	//Неисправности
	#T_notON_TON(
	             IN := (#sigOut AND NOT #OnSig AND NOT #Reset),
	             PT := #Set_T_notON
	);
	
	#notON := (#notON OR #T_notON_TON.Q) AND NOT #Reset;
	
	#T_notOFF_TON(
	             IN := (NOT #sigOut AND #OnSig AND NOT #Reset),
	             PT := #Set_T_notOFF
	);
	
	#notOFF := (#notOFF OR #T_notOFF_TON.Q) AND NOT #Reset;
	
	
	//Обобщенная неисправность
	#Fault := #notON OR #notOFF;
	
	//Авария
	#Alarm := (#Alarm OR #OnSig AND #sigOut AND NOT #Ready) AND NOT (#Reset);
	
	IF #DU THEN
	    #setSpeed := #setSpeedDU;
	ELSE
	    #setSpeed := #setSpeedAU;
	END_IF;
	
	#btnDU := false;
	
END_FUNCTION_BLOCK

FUNCTION_BLOCK "FB_IM1x1"
{ S7_Optimized_Access := 'FALSE' }
AUTHOR : Ivanez
VERSION : 0.1
//Абстактный механизм с 1й командой, 1й обратной связью (АУ, ДУ, МУ)
   VAR_INPUT 
      OnSig : Bool;   //      Сигнал сработавшего состояния
      OnCom : Bool;   //      Команда включения в автоматическом режиме
      Ready : Bool;   //      Условие готовности
      Reset : Bool;   //      Сброс
      btnAU : Bool;   //      Перевести в Автоматическое управление
      btnDU : Bool;   //      Перевести в Дистанционное управление
      prmDU : Bool;   //      Разрешение на перевод в ДУ
      btnDU_ON : Bool;   //      Включить в дистанционном управлении
      btnDU_OF : Bool;   //      Отключить в дистанционном управлении
      btnMU : Bool;   //      Перевести в местное управление
      btnMU_ON : Bool;   //      Включить в местном управлении
      btnMU_OF : Bool;   //      Отключить в местном управлении
      Set_T_notON : Time;   //      Задержа на формирование невключения
      Set_T_notOFF : Time;   //      Задержа на формирование неотключения
      setSpeedAU : Real;   //      Скорость в режиме автомат
      setSpeedDU : Real;   //      Скорость в режиме ДУoutputs
   END_VAR

   VAR_OUTPUT 
      AU : Bool;   //      Автоматическое управление (АУ)
      DU : Bool;   //      Дистанционное управление (ДУ)
      MU : Bool;   //      Местное управление (ДУ)
      notON : Bool;   //      Предупреждение о невключении
      notOFF : Bool;   //      Предупреждение о неотключении
      Alarm : Bool;   //      Авария (исчезновение готовности при работе)
      Fault : Bool;   //      Неисправность
      onOutFWD : Bool;   //      Сигнал на сработку механизма вперед
      PRM_btnDU_ON : Bool;   //      Разрешение кнопки включения в ДУ
      PRM_btnDU_OFF : Bool;   //      Разрешение кнопки отключения в ДУ
      setSpeed : Real;   //      скорость в автомате для частотникаvariables
   END_VAR

   VAR 
      sigOut : Bool;   //      Сигнал включения
      T_notON_TON {InstructionName := 'TON'; LibVersion := '1.0'; S7_SetPoint := 'False'} : TON;   //      Таймер невключения
      T_notOFF_TON {InstructionName := 'TON'; LibVersion := '1.0'; S7_SetPoint := 'False'} : TON;   //      Таймер неотключения
   END_VAR


BEGIN
	
	//Формирование автоматического управления
	IF #btnAU THEN
	    #AU := true;
	    #DU := false;
	    #MU := false;
	END_IF;
	//Формирование дистанционного управления 
	IF #btnDU THEN
	    #DU := true;
	    #AU := false;
	    #MU := false;
	END_IF;
	//Формирование местного управления
	IF #btnMU THEN
	    #MU := true;
	    #AU := false;
	    #DU := false;
	END_IF;
	
	IF NOT #AU AND NOT #DU AND NOT #MU THEN
	    #MU := true;
	END_IF;
	
	
	//Разрешения кнопок управления
	#PRM_btnDU_ON := (NOT #OnSig AND #DU OR #notON);
	#PRM_btnDU_OFF := ((#sigOut OR #OnSig) AND #DU OR #notOFF);
	
	
	//Формирование выходного сигнала
	#sigOut := #Ready AND ((#sigOut
	OR #AU AND #OnCom
	OR #DU AND #btnDU_ON
	OR #MU AND #btnMU_ON
	)
	AND NOT
	(#Alarm
	OR #AU AND NOT #OnCom
	OR #DU AND #btnDU_OF
	OR #MU AND #btnMU_OF
	OR #notON));
	
	#onOutFWD := #sigOut;
	
	//Неисправности
	#T_notON_TON(IN := (#sigOut AND NOT #OnSig AND NOT #Reset),
	             PT := #Set_T_notON
	);
	#notON := (#notON OR #T_notON_TON.Q) AND NOT #Reset;
	
	#T_notOFF_TON(IN := (NOT #sigOut AND #OnSig AND NOT #Reset),
	              PT := #Set_T_notOFF
	);
	#notOFF := (#notOFF OR #T_notOFF_TON.Q) AND NOT #Reset;
	
	//Обобщенная неисправность
	#Fault := #notON OR #notOFF;
	
	//Авария
	#Alarm := (#Alarm OR #OnSig AND #sigOut AND NOT #Ready) AND NOT (#Reset);
	
	IF #DU THEN
	    #setSpeed := #setSpeedDU;
	ELSE
	    #setSpeed := #setSpeedAU;
	END_IF;
	
END_FUNCTION_BLOCK

FUNCTION_BLOCK "FB_IM_Rout"
{ S7_Optimized_Access := 'FALSE' }
VERSION : 0.1
   VAR 
      M_321_Rollgang_Lift_PFM { S7_SetPoint := 'False'} : "FB_IM2x1";   // выкатной транспортер на лифте ПФМки
      M_322_Conveyor_2 : "FB_IM2x1";   // Выкатной транспортер после лифта
      M_324_Rout_Conveyor : "FB_IM2x1";   // выкатной транспортер последний
   END_VAR


BEGIN
	#M_321_Rollgang_Lift_PFM(OnSig:="DGI".F321K1_321K2,
	                         Ready:="ALG".Ready_Rout,
	                         Reset:="ALG".Reset OR "DGI".S76_2,
	                         btnAU:="ServDB".M_321.BtnAU OR "ALG".Auto_Sorting,
	                         btnDU:= "ServDB".M_321.BtnDU,
	                         prmDU:=TRUE,
	                         btnDU_ON:="ServDB".M_321.BtnFwd OR "ServDB".M_321.BtnBwd,
	                         btnDU_OF:="ServDB".M_321.BtnCmdStop,
	                         btnMU:="DGI".E88_3 OR "DGI".S88_2,
	                         btnMU_ON:="DGI".E88_3 OR "DGI".S88_2,
	                         btnMU_OF:=NOT ("DGI".E88_3 OR "DGI".S88_2),
	                         btn_Back_ON:= "ServDB".M_321.BtnBwd OR "DGI".S88_2,
	                         btn_Back_OFF:=NOT ("ServDB".M_321.BtnBwd OR "DGI".S88_2),
	                         Set_T_notON:=T#500ms,
	                         Set_T_notOFF:=T#500ms,
	                         AU=>"ServDB".M_321.AU,
	                         DU=>"ServDB".M_321.DU,
	                         MU=>"ServDB".M_321.MU,
	                         BACK=>"ServDB".M_321.BACK,
	                         Alarm=>"ServDB".M_321.Alarm,
	                         Fault=>"ServDB".M_321.Fault,
	                         onOutFWD=>"ServDB".M_321.CMD_ON,
	                         onOutBWD=>"ServDB".M_321.CMD_OFF,
	                         PRM_btnDU_ON=>"ServDB".M_321.PrmBtnDU_ON,
	                         PRM_btnDU_OFF=>"ServDB".M_321.PrmBtnDU_OF,
	                         PRMbtn_Back_ON=>"ServDB".M_321.PRMbtn_Back_ON,
	                         PRMbtn_Back_OFF=>"ServDB".M_321.PRMbtn_Back_OFF,
	                         setSpeed=>"ServDB".M_321.SetSpeed
	);
	
	"K1-321X1" := #M_321_Rollgang_Lift_PFM.onOutFWD AND "DGI".S16_1;
	"K1-321X1.1" := #M_321_Rollgang_Lift_PFM.onOutBWD AND "DGI".S16_1;
	
	
	
	#M_322_Conveyor_2(OnSig:="DGI".F322K1_322K2,
	                  Ready:="ALG".Ready_Rout,
	                  Reset:="ALG".Reset OR "DGI".S76_2,
	                  btnAU:="ServDB".M_322.BtnAU OR "ALG".Auto_Sorting,
	                  btnDU:="ServDB".M_322.BtnDU,
	                  prmDU:=TRUE,
	                  btnDU_ON:="ServDB".M_322.BtnFwd OR "ServDB".M_322.BtnBwd,
	                  btnDU_OF:="ServDB".M_322.BtnCmdStop,
	                  btnMU:= "DGI".S88_5 OR "DGI".S88_4,
	                  btnMU_ON:="DGI".S88_5 OR "DGI".S88_4,
	                  btnMU_OF:=NOT ("DGI".S88_5 OR "DGI".S88_4),
	                  btn_Back_ON:="ServDB".M_322.BtnBwd OR "DGI".S88_4,
	                  btn_Back_OFF:=NOT ("ServDB".M_322.BtnBwd OR "DGI".S88_4),
	                  Set_T_notON:=T#500ms,
	                  Set_T_notOFF:=T#500ms,
	                  AU=>"ServDB".M_322.AU,
	                  DU=>"ServDB".M_322.DU,
	                  MU=>"ServDB".M_322.MU,
	                  BACK=>"ServDB".M_322.BACK,
	                  Alarm=>"ServDB".M_322.Alarm,
	                  Fault=>"ServDB".M_322.Fault,
	                  onOutFWD=>"ServDB".M_322.CMD_ON,
	                  onOutBWD=>"ServDB".M_322.CMD_OFF,
	                  PRM_btnDU_ON=>"ServDB".M_322.PrmBtnDU_ON,
	                  PRM_btnDU_OFF=>"ServDB".M_322.PrmBtnDU_OF,
	                  PRMbtn_Back_ON=>"ServDB".M_322.PRMbtn_Back_ON,
	                  PRMbtn_Back_OFF=>"ServDB".M_322.PRMbtn_Back_OFF,
	                  setSpeed=>"ServDB".M_322.SetSpeed
	);
	
	
	"K1-322X1" := #M_322_Conveyor_2.onOutFWD;
	"K1-322X1.1" := #M_322_Conveyor_2.onOutBWD;
	
	#M_324_Rout_Conveyor(OnSig:="DGI".K1_324U1,
	                     Ready:="ALG".Ready_Rout,
	                     Reset:="ALG".Reset OR "DGI".S76_2,
	                     btnAU:= "ServDB".M_324.BtnAU OR "ALG".Auto_Sorting,
	                     btnDU:= "ServDB".M_324.BtnDU,
	                     prmDU:=TRUE,
	                     btnDU_ON:="ServDB".M_324.BtnFwd OR "ServDB".M_324.BtnBwd,
	                     btnDU_OF:="ServDB".M_324.BtnCmdStop,
	                     btnMU:= "DGI".S89_1 OR "DGI".S89_0,
	                     btnMU_ON:="DGI".S89_1 OR "DGI".S89_0,
	                     btnMU_OF:=NOT ("DGI".S89_1 OR "DGI".S89_0),
	                     btn_Back_ON:= "DGI".S89_0 OR "ServDB".M_324.BtnBwd,
	                     btn_Back_OFF:=NOT ("DGI".S89_0 OR "ServDB".M_324.BtnBwd),
	                     Set_T_notON:=T#1s,
	                     Set_T_notOFF:=T#2s,
	                     AU=>"ServDB".M_324.AU,
	                     DU=>"ServDB".M_324.DU,
	                     MU=>"ServDB".M_324.MU,
	                     BACK=>"ServDB".M_324.BACK,
	                     Alarm=>"ServDB".M_324.Alarm,
	                     Fault=>"ServDB".M_324.Fault,
	                     onOutFWD=>"ServDB".M_324.CMD_ON,
	                     onOutBWD=>"ServDB".M_324.CMD_OFF,
	                     PRM_btnDU_ON=>"ServDB".M_324.PrmBtnDU_ON,
	                     PRM_btnDU_OFF=>"ServDB".M_324.PrmBtnDU_OF,
	                     PRMbtn_Back_ON=>"ServDB".M_324.PRMbtn_Back_ON,
	                     PRMbtn_Back_OFF=>"ServDB".M_324.PRMbtn_Back_OFF,
	                     setSpeed=>"ServDB".M_324.SetSpeed
	);
	
	"K1-324U2" := #M_324_Rout_Conveyor.onOutFWD;
	"K1-324U2.2" := #M_324_Rout_Conveyor.onOutBWD;
	
END_FUNCTION_BLOCK

ORGANIZATION_BLOCK "PROG_ERR"   // OB121, LAD, ProgrammingError
TITLE = "Programming Error"
VERSION : 0.1
// stored: IsIECCheckEnabled false
   VAR_TEMP
      OB121_EV_CLASS : Byte;   // 16#25, Event class 2, Entering event state, Internal fault event
      OB121_SW_FLT : Byte;   // 16#XX Software programming fault
      OB121_PRIORITY : Byte;   // Priority of OB Execution
      OB121_OB_NUMBR : Byte;   // 121 (Organization block 121, OB121)
      OB121_BLK_TYPE : Byte;   // 16#88/8A/8B/8C/8E Type of block fault occured in
      OB121_RESERVED_1 : Byte;   // Reserved for system
      OB121_FLT_REG : Word;   // 16#XX Specific register that caused fault
      OB121_BLK_NUM : Word;   // Number of block that programming fault occured in
      OB121_PRG_ADDR : Word;   // Address in block where programming fault occured
      OB121_DATE_TIME : Date_And_Time;   // Date and time OB121 started
   END_VAR
BEGIN
END_ORGANIZATION_BLOCK

ORGANIZATION_BLOCK "BREAKUP ERROR"   // OB88, LAD, ProcessingInterrupt
TITLE = "Breakup Error"
VERSION : 0.1
// stored: IsIECCheckEnabled false
   VAR_TEMP
      OB88_EV_CLASS : Byte;   // 16#35 Event class 2, Entering event state, Internal fault event
      OB88_SW_FLT : Byte;   // 16#XX, Software programming fault
      OB88_PRIORITY : Byte;   // Priority of OB Execution
      OB88_OB_NUMBR : Byte;   // 88 (Organization block 88, OB88)
      OB88_BLK_TYPE : Byte;   // 16#88/8C/8E Type of block where breakup occured
      OB88_RESERVED_1 : Byte;   // Reserved for system
      OB88_FLT_PRIORITY : Byte;   // Priority of OB caused breakup
      OB88_FLT_OB_NUMBR : Byte;   // OB execution caused breakup
      OB88_BLK_NUM : Word;   // Number of block where breakup occured
      OB88_PRG_ADDR : Word;   // Address in block where breakup occured
      OB88_DATE_TIME : Date_And_Time;   // Date and time OB88 started
   END_VAR
BEGIN
END_ORGANIZATION_BLOCK

ORGANIZATION_BLOCK "COMM_FLT"   // OB87, LAD, CommunicationError
TITLE = "Communication Fault"
VERSION : 0.1
// stored: IsIECCheckEnabled false
   VAR_TEMP
      OB87_EV_CLASS : Byte;   // 16#39 Event class 3
      OB87_FLT_ID : Byte;   // 16#XX, Fault identifcation code
      OB87_PRIORITY : Byte;   // Priority of OB Execution
      OB87_OB_NUMBR : Byte;   // 87 (Organization block 87, OB87)
      OB87_RESERVED_1 : Byte;   // Reserved for system
      OB87_RESERVED_2 : Byte;   // Reserved for system
      OB87_RESERVED_3 : Word;   // Reserved for system
      OB87_RESERVED_4 : DWord;   // Reserved for system
      OB87_DATE_TIME : Date_And_Time;   // Date and time OB87 started
   END_VAR
BEGIN
END_ORGANIZATION_BLOCK

ORGANIZATION_BLOCK "CPU_FLT"   // OB84, LAD, CPUHardwareError
TITLE = "CPU Fault"
VERSION : 0.1
// stored: IsIECCheckEnabled false
   VAR_TEMP
      OB84_EV_CLASS : Byte;   // 16#38/39, Event class 3, module inserted/removed (8/9)
      OB84_FLT_ID : Byte;   // 16#81, Fault identifcation code
      OB84_PRIORITY : Byte;   // Priority of OB Execution
      OB84_OB_NUMBR : Byte;   // 84 (Organization block 84, OB84)
      OB84_RESERVED_1 : Byte;   // Reserved for system
      OB84_RESERVED_2 : Byte;   // Reserved for system
      OB84_RESERVED_3 : Word;   // Reserved for system
      OB84_RESERVED_4 : DWord;   // Reserved for system
      OB84_DATE_TIME : Date_And_Time;   // Date and time OB84 started
   END_VAR
BEGIN
END_ORGANIZATION_BLOCK

ORGANIZATION_BLOCK "CYCL_FLT"   // OB80, LAD, TimeErrorInterrupt
TITLE = "Cycle Time Fault"
VERSION : 0.1
// stored: IsIECCheckEnabled false
   VAR_TEMP
      OB80_EV_CLASS : Byte;   // 16#35, Event class 3, Entering event state, Internal fault event
      OB80_FLT_ID : Byte;   // 16#XX, Fault identifcation code
      OB80_PRIORITY : Byte;   // Priority of OB Execution
      OB80_OB_NUMBR : Byte;   // 80 (Organization block 80, OB80)
      OB80_RESERVED_1 : Byte;   // Reserved for system
      OB80_RESERVED_2 : Byte;   // Reserved for system
      OB80_ERROR_INFO : Word;   // Error information on event
      OB80_ERR_EV_CLASS : Byte;   // Class of event causing error
      OB80_ERR_EV_NUM : Byte;   // Number of event causing error
      OB80_OB_PRIORITY : Byte;   // Priority of OB causing error
      OB80_OB_NUM : Byte;   // Number of OB causing error
      OB80_DATE_TIME : Date_And_Time;   // Date and time OB80 started
   END_VAR
BEGIN
END_ORGANIZATION_BLOCK

ORGANIZATION_BLOCK "MOD_ERR"   // OB122, LAD, IOAccessError
TITLE = "Module Access Error"
VERSION : 0.1
// stored: IsIECCheckEnabled false
   VAR_TEMP
      OB122_EV_CLASS : Byte;   // 16#29, Event class 2, Entering event state, Internal fault event
      OB122_SW_FLT : Byte;   // 16#XX Software error code
      OB122_PRIORITY : Byte;   // Priority of OB Execution
      OB122_OB_NUMBR : Byte;   // 122 (Organization block 122, OB122)
      OB122_BLK_TYPE : Byte;   // 16#88/8C/8E Type of block fault occured in
      OB122_MEM_AREA : Byte;   // Memory area where access error occured
      OB122_MEM_ADDR : Word;   // Memory address where access error occured
      OB122_BLK_NUM : Word;   // Block number in which error occured
      OB122_PRG_ADDR : Word;   // Program address where error occured
      OB122_DATE_TIME : Date_And_Time;   // Date and time OB1 started
   END_VAR
BEGIN
END_ORGANIZATION_BLOCK

ORGANIZATION_BLOCK "OBNL_FLT"   // OB85, LAD, AccessError
TITLE = "Organization Block (OB) Not Loaded Fault"
VERSION : 0.1
// stored: IsIECCheckEnabled false
   VAR_TEMP
      OB85_EV_CLASS : Byte;   // 16#35 Event class 3
      OB85_FLT_ID : Byte;   // 16#XX, Fault identification code
      OB85_PRIORITY : Byte;   // Priority of OB Execution
      OB85_OB_NUMBR : Byte;   // 85 (Organization block 85, OB85)
      OB85_RESERVED_1 : Byte;   // Reserved for system
      OB85_RESERVED_2 : Byte;   // Reserved for system
      OB85_RESERVED_3 : Int;   // Reserved for system
      OB85_ERR_EV_CLASS : Byte;   // Class of event causing error
      OB85_ERR_EV_NUM : Byte;   // Number of event causing error
      OB85_OB_PRIOR : Byte;   // Priority of OB causing error
      OB85_OB_NUM : Byte;   // Number of OB causing error
      OB85_DATE_TIME : Date_And_Time;   // Date and time OB85 started
   END_VAR
BEGIN
END_ORGANIZATION_BLOCK

ORGANIZATION_BLOCK "PS_FLT"   // OB81, LAD, PowerSupplyError
TITLE = "Power Supply Fault"
VERSION : 0.1
// stored: IsIECCheckEnabled false
   VAR_TEMP
      OB81_EV_CLASS : Byte;   // 16#39, Event class 3, Entering event state, Internal fault event
      OB81_FLT_ID : Byte;   // 16#XX, Fault identifcation code
      OB81_PRIORITY : Byte;   // Priority of OB Execution
      OB81_OB_NUMBR : Byte;   // 81 (Organization block 81, OB81)
      OB81_RESERVED_1 : Byte;   // Reserved for system
      OB81_RESERVED_2 : Byte;   // Reserved for system
      OB81_RACK_CPU : Word;   // Bits 0 to 2: Rack no; Bit 3: 0=standby CPU, 1=master CPU; Bits 4 to 7: 1111
      OB81_RESERVED_3 : Byte;   // Reserved for system
      OB81_RESERVED_4 : Byte;   // Reserved for system
      OB81_RESERVED_5 : Byte;   // Reserved for system
      OB81_RESERVED_6 : Byte;   // Reserved for system
      OB81_DATE_TIME : Date_And_Time;   // Date and time OB81 started
   END_VAR
BEGIN
END_ORGANIZATION_BLOCK

ORGANIZATION_BLOCK "RACK_FLT"   // OB86, LAD, RackOrStationFailure
TITLE = "Loss Of Rack Fault"
VERSION : 0.1
// stored: IsIECCheckEnabled false
   VAR_TEMP
      OB86_EV_CLASS : Byte;   // 16#38/39 Event class 3
      OB86_FLT_ID : Byte;   // 16#C1/C4/C5, Fault identification code
      OB86_PRIORITY : Byte;   // Priority of OB Execution
      OB86_OB_NUMBR : Byte;   // 86 (Organization block 86, OB86)
      OB86_RESERVED_1 : Byte;   // Reserved for system
      OB86_RESERVED_2 : Byte;   // Reserved for system
      OB86_MDL_ADDR : Word;   // Base address of IM module in rack with fault
      OB86_RACKS_FLTD : Array[0..31] of Bool;   // Racks in fault
      OB86_DATE_TIME : Date_And_Time;   // Date and time OB86 started
   END_VAR
BEGIN
END_ORGANIZATION_BLOCK

FUNCTION_BLOCK "Загрузка"   // FB8, LAD
VERSION : 0.1
// stored: AutoNumber true, IsIECCheckEnabled false, UDAEnableTagReadback false
   VAR DB_SPECIFIC
      "TrigS84.4" : Bool;
      LiftUpTrig : Bool;
      "212StartCNTL" : Bool;
      "TrigS82.3/S76.5" : Bool;
      LiftDownTrig : Bool;
   END_VAR
   VAR_TEMP
      Sert : Word;
      AutoLamp : Bool;
      M213_wide_mode : Bool;
   END_VAR
   VAR_TEMP   // added for the SCL form of the ladder/FBD networks
      _w1 : Bool;
      _s5time1 : S5Time;
      _w2 : Bool;
      _w3 : Bool;
      _w4 : Bool;
      _s5time2 : S5Time;
   END_VAR
BEGIN

REGION Network 1: 211 группа на 4 мотора обющий сигнал готовности
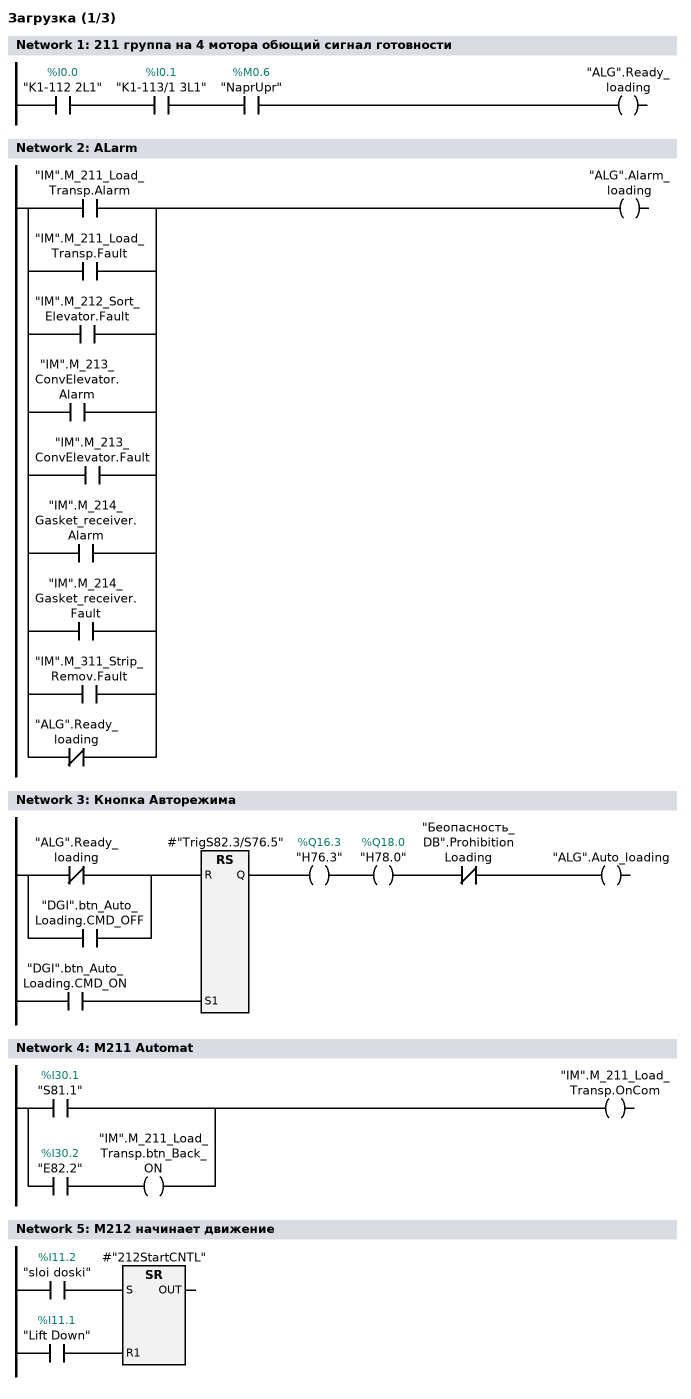
   RUNG wire#powerrail
      Contact( "K1-112 2L1" )
      Contact( "K1-113/1 3L1" )
      Contact( "NaprUpr" )
      Coil( "ALG".Ready_loading )
   END_RUNG
   // the same network as SCL:
   "ALG".Ready_loading := "K1-112 2L1" AND "K1-113/1 3L1" AND "NaprUpr";
END_REGION

REGION Network 2: ALarm
   RUNG wire#powerrail
      Contact( "IM".M_211_Load_Transp.Alarm )
      wire#w1
      Coil( "ALG".Alarm_loading )
   END_RUNG
   RUNG wire#powerrail
      Contact( "IM".M_211_Load_Transp.Fault )
   END_RUNG wire#w1
   RUNG wire#powerrail
      Contact( "IM".M_212_Sort_Elevator.Fault )
   END_RUNG wire#w1
   RUNG wire#powerrail
      Contact( "IM".M_213_ConvElevator.Alarm )
   END_RUNG wire#w1
   RUNG wire#powerrail
      Contact( "IM".M_213_ConvElevator.Fault )
   END_RUNG wire#w1
   RUNG wire#powerrail
      Contact( "IM".M_214_Gasket_receiver.Alarm )
   END_RUNG wire#w1
   RUNG wire#powerrail
      Contact( "IM".M_214_Gasket_receiver.Fault )
   END_RUNG wire#w1
   RUNG wire#powerrail
      Contact( "IM".M_311_Strip_Remov.Fault )
   END_RUNG wire#w1
   RUNG wire#powerrail
      I_Contact( "ALG".Ready_loading )
   END_RUNG wire#w1
   // the same network as SCL:
   "ALG".Alarm_loading := "IM".M_211_Load_Transp.Alarm OR "IM".M_211_Load_Transp.Fault OR "IM".M_212_Sort_Elevator.Fault OR "IM".M_213_ConvElevator.Alarm OR "IM".M_213_ConvElevator.Fault OR "IM".M_214_Gasket_receiver.Alarm OR "IM".M_214_Gasket_receiver.Fault OR "IM".M_311_Strip_Remov.Fault OR NOT "ALG".Ready_loading;
END_REGION

REGION Network 3: Кнопка Авторежима
   RUNG wire#powerrail
      I_Contact( "ALG".Ready_loading )
      wire#w1
      S_RS(operand := #"TrigS82.3/S76.5", s1 := wire#w2)
      Coil( "H76.3" )
      Coil( "H78.0" )
      I_Contact( "Беопасность_DB".ProhibitionLoading )
      Coil( "ALG".Auto_loading )
   END_RUNG
   RUNG wire#powerrail
      Contact( "DGI".btn_Auto_Loading.CMD_OFF )
   END_RUNG wire#w1
   RUNG wire#powerrail
      Contact( "DGI".btn_Auto_Loading.CMD_ON )
   END_RUNG wire#w2
   // the same network as SCL:
   IF NOT "ALG".Ready_loading OR "DGI".btn_Auto_Loading.CMD_OFF THEN
       #"TrigS82.3/S76.5" := FALSE;   // RS flip-flop
   END_IF;
   IF "DGI".btn_Auto_Loading.CMD_ON THEN #"TrigS82.3/S76.5" := TRUE; END_IF;
   "H76.3" := #"TrigS82.3/S76.5";
   "H78.0" := #"TrigS82.3/S76.5";
   "ALG".Auto_loading := #"TrigS82.3/S76.5" AND NOT "Беопасность_DB".ProhibitionLoading;
END_REGION

REGION Network 4: M211 Automat
   RUNG wire#powerrail
      Contact( "S81.1" )
      wire#w1
      Coil( "IM".M_211_Load_Transp.OnCom )
   END_RUNG
   RUNG wire#powerrail
      Contact( "E82.2" )
      Coil( "IM".M_211_Load_Transp.btn_Back_ON )
   END_RUNG wire#w1
   // the same network as SCL:
   "IM".M_211_Load_Transp.btn_Back_ON := "E82.2";
   "IM".M_211_Load_Transp.OnCom := "S81.1" OR "E82.2";
END_REGION

REGION Network 5: M212 начинает движение
   RUNG wire#powerrail
      Contact( "sloi doski" )
      S_SR(operand := #"212StartCNTL", r1 := wire#w1)
   END_RUNG
   RUNG wire#powerrail
      Contact( "Lift Down" )
   END_RUNG wire#w1
   // the same network as SCL:
   IF "sloi doski" THEN
       #"212StartCNTL" := TRUE;   // SR flip-flop
   END_IF;
   IF "Lift Down" THEN #"212StartCNTL" := FALSE; END_IF;
END_REGION

REGION Network 6: М212 AutoMode
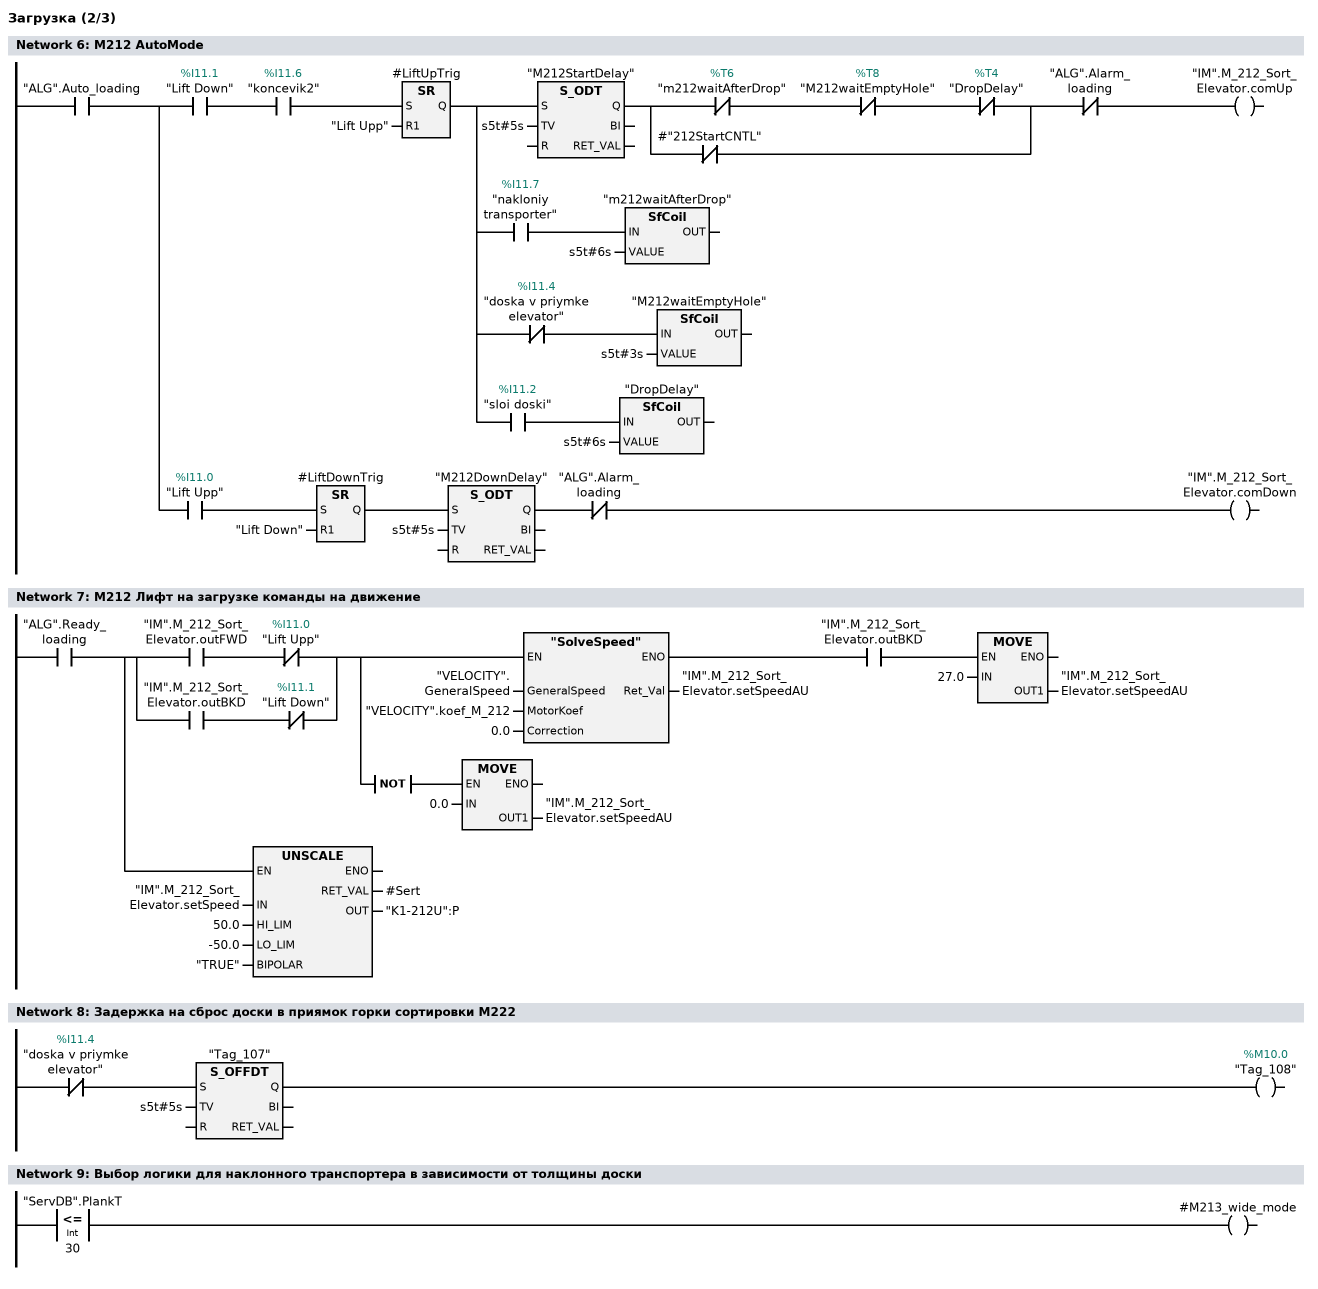
   // no SCL statement known for SfCoil: written as a call
   IF "ALG".Auto_loading AND "Lift Down" AND "koncevik2" THEN
       #LiftUpTrig := TRUE;   // SR flip-flop
   END_IF;
   IF "Lift Upp" THEN #LiftUpTrig := FALSE; END_IF;
   #_w2 := #LiftUpTrig;
   #_s5time1 := S_ODT(T_NO := "M212StartDelay", S := #LiftUpTrig, TV := s5t#5s, Q => #_w1);
   "IM".M_212_Sort_Elevator.comUp := #_w1 AND ((NOT "m212waitAfterDrop" AND NOT "M212waitEmptyHole" AND NOT "DropDelay") OR NOT #"212StartCNTL") AND NOT "ALG".Alarm_loading;
   #_w3 := "ALG".Auto_loading;
   SfCoil(in := #_w2 AND "nakloniy transporter", value := s5t#6s, operand := "m212waitAfterDrop");
   SfCoil(in := #_w2 AND NOT "doska v priymke elevator", value := s5t#3s, operand := "M212waitEmptyHole");
   SfCoil(in := #_w2 AND "sloi doski", value := s5t#6s, operand := "DropDelay");
   IF #_w3 AND "Lift Upp" THEN
       #LiftDownTrig := TRUE;   // SR flip-flop
   END_IF;
   IF "Lift Down" THEN #LiftDownTrig := FALSE; END_IF;
   #_s5time2 := S_ODT(T_NO := "M212DownDelay", S := #LiftDownTrig, TV := s5t#5s, Q => #_w4);
   "IM".M_212_Sort_Elevator.comDown := #_w4 AND NOT "ALG".Alarm_loading;
END_REGION

REGION Network 7: М212 Лифт на загрузке команды на движение
   RUNG wire#powerrail
      Contact( "ALG".Ready_loading )
      wire#w1
      Contact( "IM".M_212_Sort_Elevator.outFWD )
      I_Contact( "Lift Upp" )
      wire#w2
      "SolveSpeed"(GeneralSpeed := "VELOCITY".GeneralSpeed, MotorKoef := "VELOCITY".koef_M_212, Correction := 0.0, Ret_Val => "IM".M_212_Sort_Elevator.setSpeedAU)
      Contact( "IM".M_212_Sort_Elevator.outBKD )
      { S7_GenerateENO := "TRUE" } Move(in := 27.0, out1 => "IM".M_212_Sort_Elevator.setSpeedAU)
   END_RUNG
   RUNG wire#w1
      Contact( "IM".M_212_Sort_Elevator.outBKD )
      I_Contact( "Lift Down" )
   END_RUNG wire#w2
   RUNG wire#w2
      Not()
      { S7_GenerateENO := "TRUE" } Move(in := 0.0, out1 => "IM".M_212_Sort_Elevator.setSpeedAU)
   END_RUNG
   RUNG wire#w1
      UNSCALE(IN := "IM".M_212_Sort_Elevator.setSpeed, HI_LIM := 50.0, LO_LIM := -50.0, BIPOLAR := "TRUE", RET_VAL => #Sert, OUT => "K1-212U":P)
   END_RUNG
   // the same network as SCL:
   #_w1 := "ALG".Ready_loading AND (("IM".M_212_Sort_Elevator.outFWD AND NOT "Lift Upp") OR ("IM".M_212_Sort_Elevator.outBKD AND NOT "Lift Down"));
   #_w3 := "ALG".Ready_loading;
   "IM".M_212_Sort_Elevator.setSpeedAU := "SolveSpeed"(EN := #_w1,
                           GeneralSpeed := "VELOCITY".GeneralSpeed,
                           MotorKoef := "VELOCITY".koef_M_212,
                           Correction := 0.0,
                           ENO => #_w2);
   IF #_w2 AND "IM".M_212_Sort_Elevator.outBKD THEN "IM".M_212_Sort_Elevator.setSpeedAU := 27.0; END_IF;
   IF NOT #_w1 THEN "IM".M_212_Sort_Elevator.setSpeedAU := 0.0; END_IF;
   IF #_w3 THEN
       #Sert := UNSCALE(IN := "IM".M_212_Sort_Elevator.setSpeed,
                        HI_LIM := 50.0,
                        LO_LIM := -50.0,
                        BIPOLAR := "TRUE",
                        OUT => "K1-212U":P);
   END_IF;
END_REGION

REGION Network 8: Задержка на сброс доски в приямок горки сортировки М222
   RUNG wire#powerrail
      I_Contact( "doska v priymke elevator" )
      S_OFFDT(T_NO := "Tag_107", TV := s5t#5s, R :=, BI =>, RET_VAL =>)
      Coil( "Tag_108" )
   END_RUNG
   // the same network as SCL:
   #_s5time1 := S_OFFDT(T_NO := "Tag_107", S := NOT "doska v priymke elevator", TV := s5t#5s, Q => #_w1);
   "Tag_108" := #_w1;
END_REGION

REGION Network 9: Выбор логики для наклонного транспортера в зависимости от толщины доски
   RUNG wire#powerrail
      { S7_Templates := "SrcType := Int" } LE_Contact(in1 := "ServDB".PlankT, in2 := 30)
      Coil( #M213_wide_mode )
   END_RUNG
   // the same network as SCL:
   #M213_wide_mode := "ServDB".PlankT <= 30;
END_REGION

REGION Network 10: М213 Наклонный транспортер Авто вперед
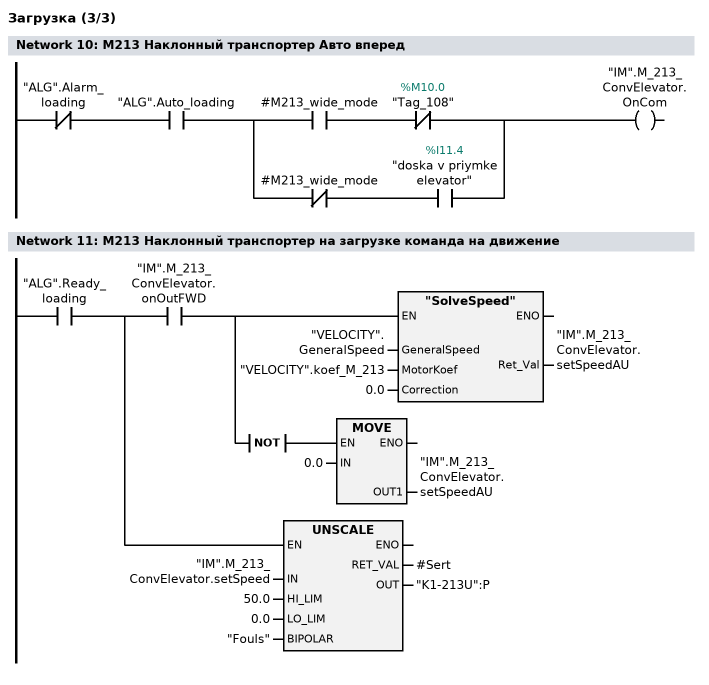
   RUNG wire#powerrail
      I_Contact( "ALG".Alarm_loading )
      Contact( "ALG".Auto_loading )
      wire#w1
      Contact( #M213_wide_mode )
      I_Contact( "Tag_108" )
      wire#w2
      Coil( "IM".M_213_ConvElevator.OnCom )
   END_RUNG
   RUNG wire#w1
      I_Contact( #M213_wide_mode )
      Contact( "doska v priymke elevator" )
   END_RUNG wire#w2
   // the same network as SCL:
   "IM".M_213_ConvElevator.OnCom := NOT "ALG".Alarm_loading AND "ALG".Auto_loading AND ((#M213_wide_mode AND NOT "Tag_108") OR (NOT #M213_wide_mode AND "doska v priymke elevator"));
END_REGION

REGION Network 11: М213 Наклонный транспортер на загрузке команда на движение
   RUNG wire#powerrail
      Contact( "ALG".Ready_loading )
      wire#w1
      Contact( "IM".M_213_ConvElevator.onOutFWD )
      wire#w2
      "SolveSpeed"(GeneralSpeed := "VELOCITY".GeneralSpeed, MotorKoef := "VELOCITY".koef_M_213, Correction := 0.0, Ret_Val => "IM".M_213_ConvElevator.setSpeedAU)
   END_RUNG
   RUNG wire#w2
      Not()
      { S7_GenerateENO := "TRUE" } Move(in := 0.0, out1 => "IM".M_213_ConvElevator.setSpeedAU)
   END_RUNG
   RUNG wire#w1
      UNSCALE(IN := "IM".M_213_ConvElevator.setSpeed, HI_LIM := 50.0, LO_LIM := 0.0, BIPOLAR := "Fouls", RET_VAL => #Sert, OUT => "K1-213U":P)
   END_RUNG
   // the same network as SCL:
   #_w1 := "ALG".Ready_loading AND "IM".M_213_ConvElevator.onOutFWD;
   #_w2 := "ALG".Ready_loading;
   IF #_w1 THEN
       "IM".M_213_ConvElevator.setSpeedAU := "SolveSpeed"(GeneralSpeed := "VELOCITY".GeneralSpeed,
                               MotorKoef := "VELOCITY".koef_M_213,
                               Correction := 0.0);
   END_IF;
   IF NOT #_w1 THEN "IM".M_213_ConvElevator.setSpeedAU := 0.0; END_IF;
   IF #_w2 THEN
       #Sert := UNSCALE(IN := "IM".M_213_ConvElevator.setSpeed,
                        HI_LIM := 50.0,
                        LO_LIM := 0.0,
                        BIPOLAR := "Fouls",
                        OUT => "K1-213U":P);
   END_IF;
END_REGION
END_FUNCTION_BLOCK

FUNCTION_BLOCK "Button_Clicker_LongTap"
{ S7_Optimized_Access := 'FALSE' }
VERSION : 0.1
   VAR_INPUT 
      Button_Sig : Bool;   //  сигнал с кнопки
      set_Trembling_Time : Time;   //  время на дребезг контактов
      set_LongTapFixation_Time : Time;   //  время ожидания долгого тапа
   END_VAR

   VAR_OUTPUT 
      CMD_ON : Bool;   //  сигнал включения
      CMD_Double : Bool;   // сигнал двойного клика
      CMD_Triple : Bool;   // сигнал тройного клика
      CMD_LongTap : Bool;   //  сигнал долго нажатия
   END_VAR

   VAR 
      Timer_LongTap_old : Bool;   //  сигнал с таймера на прошлой итерации
      ClickCounter : Int;   // счет кликов кнопки
      LongTap_Timer {InstructionName := 'TON'; LibVersion := '1.0'} : TON;   //  таймер долгого нажатия
   END_VAR


BEGIN
	#CMD_ON := FALSE;
	#CMD_LongTap := False;
	
	IF (#LongTap_Timer.ET > #set_Trembling_Time AND NOT #Button_Sig) THEN
	    #CMD_ON := TRUE;
	END_IF;
	
	#LongTap_Timer(IN := #Button_Sig,
	               PT := #set_LongTapFixation_Time
	);
	
	IF (#LongTap_Timer.Q AND NOT #Timer_LongTap_old) THEN
	    #CMD_LongTap := TRUE;
	END_IF;
	
	#Timer_LongTap_old := #LongTap_Timer.Q;
END_FUNCTION_BLOCK

ORGANIZATION_BLOCK "CYC_INT3"
TITLE = "Cyclic Interrupt"
{ S7_Optimized_Access := 'FALSE' }
VERSION : 0.1
   VAR_TEMP 
      OB33_EV_CLASS : Byte;   // Bits 0-3 = 1 (Coming event), Bits 4-7 = 1 (Event class 1)
      OB33_STRT_INF : Byte;   // 16#34 (OB 33 has started)
      OB33_PRIORITY : Byte;   // Priority of OB Execution
      OB33_OB_NUMBR : Byte;   // 33 (Organization block 33, OB33)
      OB33_RESERVED_1 : Byte;   // Reserved for system
      OB33_RESERVED_2 : Byte;   // Reserved for system
      OB33_PHS_OFFSET : Int;   // Phase offset (integer, milliseconds)
      OB33_RESERVED_3 : Int;   // Reserved for system
      OB33_EXC_FREQ : Int;   // Frequency of execution (msec)
      OB33_DATE_TIME : Date_And_Time;   // Date and time OB33 started
   END_VAR


BEGIN
	IF ("ALG".Meandr = 32000) THEN
	    "ALG".Meandr := 0;
	END_IF;
	
	// счет для различных меандров большей частоты
	// 
	"ALG".Meandr := "ALG".Meandr + 1;
	
	// герцовка для ламп и прочего барахла
	// 
	"2Hz" := NOT "2Hz";
END_ORGANIZATION_BLOCK

FUNCTION_BLOCK "DI"
{ S7_Optimized_Access := 'FALSE' }
VERSION : 0.1
   VAR_INPUT 
      in : Bool;
      stableON : Time;
      stableOFF : Time;
   END_VAR

   VAR_OUTPUT 
      out : Bool;
      fe : Bool;
      de : Bool;
   END_VAR

   VAR 
      old_out : Bool;
      onTimer {InstructionName := 'TON'; LibVersion := '1.0'; S7_SetPoint := 'False'} : TON;
      offTimer {InstructionName := 'TON'; LibVersion := '1.0'; S7_SetPoint := 'False'} : TON;
   END_VAR


BEGIN
	#onTimer(
	         IN := (#in AND NOT #out),
	         PT := #stableON
	);
	
	#offTimer(
	          IN := (NOT #in AND #out),
	          PT := #stableOFF
	);
	
	IF (#onTimer.Q) THEN
	    #old_out := FALSE;
	    #out := TRUE;
	    #de := True;
	END_IF;
	
	IF (#offTimer.Q) THEN
	    #old_out := TRUE;
	    #out := FALSE;
	    #fe := True;
	END_IF;
	
END_FUNCTION_BLOCK

FUNCTION_BLOCK "FB_Lift_PFM"
{ S7_Optimized_Access := 'FALSE' }
VERSION : 0.1
   VAR_INPUT 
      lift_upper_sensor : Bool;
      lift_down_sensor : Bool;
   END_VAR


BEGIN
END_FUNCTION_BLOCK

FUNCTION_BLOCK "LodemsRamp_CNTL"
{ S7_Optimized_Access := 'FALSE' }
AUTHOR : Aspir
VERSION : 0.1
   VAR_INPUT 
      NoGasketMode : Bool;   // режим без прокладки
      OneMoreLay : Bool;   // сигнал о необходимости еще одного слоя прокладок
      GasketLayerReady : Bool;   // можно забирать свежий слой прокладок
      MidUpPermission : Bool;   // разрешение на подъем
      SafetyForcing : Bool;   // безопасный набор
      CanGoDown : Bool;   // можно ехать вниз после отъезда крюков назад
      CanPutGaskets : Bool;
      VillStartPos : Bool;   // вилы задвинуты
      LodemsOpened : Bool;   // стаканы открыты
      PacketPicked : Bool;   // пакет выкатили, можно опускаться
      PushingPacket : Bool;   // форсирование пакета
      ToEmptyGasket : Bool;
      TopStateSensor : Bool;   // датчик верхнего положения
      MidStateSensor : Bool;   // датчик среднего положения
      LowStateSensor : Bool;   // датчик нижнего положения
      QPlanksLayers : Int;   // количество слоев
   END_VAR

   VAR_OUTPUT 
      CMD_On : Bool;   // команда вверх
      CMD_Mid : Bool;   // команда вниз
      CMD_Off : Bool;
      CMD_OpenLodems : Bool;
      CMD_CloseLodems : Bool;
      Carousel_GetRidOf : Bool;
      ResetCarouselAlgo : Bool;   // сброс алгоритма карусели
      LastLay : Bool;   // последний слой прокладок
      LayerHolded : Int;   // номер удерживаемого слоя
   END_VAR

   VAR 
      BusyGaskets : Bool;   // сейчас занят
      goDown_trig : Bool;   // триггер на движение вниз
      goUp_trig : Bool;   // триггер на движение вверх
      pushing_trig : Bool;
      nogasket_old : Bool;
   END_VAR


BEGIN
	#ResetCarouselAlgo := FALSE;
	
	#pushing_trig := #pushing_trig OR #PushingPacket;
	
	//обратная связь карусели
	#Carousel_GetRidOf := (#Carousel_GetRidOf OR (#BusyGaskets AND #MidStateSensor)) AND NOT #GasketLayerReady;
	
	//логика открытия/закрытия стаканов
	//
	#CMD_OpenLodems := (#CMD_OpenLodems OR (#CMD_Off AND #LowStateSensor)) AND NOT #MidStateSensor;
	#CMD_CloseLodems := NOT #CMD_OpenLodems;
	
	//режим без прокладки выключили
	//
	IF (NOT #NoGasketMode AND #nogasket_old) THEN
	    #CMD_On := FALSE;
	    #CMD_Mid := TRUE;
	    #CMD_Off := FALSE;
	END_IF;
	
	//если вдруг неправильно сработал счет и нужен еще слой прокладок, просто нажимаем кнопку еще один слой
	//снимем флаг последний слой и спустимся в среднее положение
	//
	IF (#LastLay AND NOT #BusyGaskets AND #OneMoreLay) THEN
	    #LastLay := FALSE;
	    // едем вниз на среднее положение
	    #CMD_On := FALSE;
	    #CMD_Mid := TRUE;
	    #CMD_Off := FALSE;
	END_IF;
	
	IF (NOT #BusyGaskets AND ((#GasketLayerReady AND #MidUpPermission) OR (#pushing_trig AND #SafetyForcing) OR #LastLay OR #NoGasketMode)) THEN
	    // поднимаем прокладочник
	    // 
	    #goUp_trig := TRUE;
	    
	    #CMD_On := TRUE;
	    #CMD_Mid := FALSE;
	    #CMD_Off := FALSE;
	    
	END_IF;
	
	IF (#TopStateSensor AND #CanGoDown AND #goUp_trig AND NOT #pushing_trig) THEN
	    // Карусель говорит что можно опускаться при этом не форсируем
	    // едем вниз на среднее положение
	    #CMD_On := FALSE;
	    #CMD_Mid := TRUE;
	    #CMD_Off := FALSE;
	    
	    #goUp_trig := FALSE;
	    
	    #BusyGaskets := TRUE;
	    
	    #LayerHolded := #LayerHolded + 1;
	    
	    #LastLay := #LayerHolded >= #QPlanksLayers - 1;
	END_IF;
	
	#goDown_trig := (#goDown_trig OR #CanPutGaskets) AND NOT (#pushing_trig);
	
	IF (#BusyGaskets AND #goDown_trig AND #VillStartPos) THEN
	    // опускаем прокладочник если есть что опускать вилы сзади и есть на то команда
	    // 
	    #CMD_On := FALSE;
	    #CMD_Mid := FALSE;
	    #CMD_Off := TRUE;
	    
	    IF (#LodemsOpened AND #LowStateSensor) THEN
	            //  прокладочник в среднее положение как только сбросили прокладку
	            // 
	            #CMD_On := FALSE;
	            #CMD_Mid := true;
	            #CMD_Off := FALSE;
	            
	            #BusyGaskets := FALSE;
	            
	            #goDown_trig := False;
	        END_IF;
	END_IF;
	
	IF (#ToEmptyGasket) THEN
	    #BusyGaskets := FALSE;
	END_IF;
	
	
	IF (#PacketPicked) THEN
	
	    #pushing_trig := FALSE;
	    #LastLay := FALSE;
	    #goDown_trig := FALSE;
	    #LayerHolded := 0;
	    #ResetCarouselAlgo := TRUE;
	    //  прокладочник в среднее положение
	    // 
	    #CMD_On := FALSE;
	    #CMD_Mid := true;
	    #CMD_Off := FALSE;
	    
	END_IF;
	
	#nogasket_old := #NoGasketMode;
END_FUNCTION_BLOCK

FUNCTION_BLOCK "SensorRuntime_checker"
{ S7_Optimized_Access := 'FALSE' }
VERSION : 0.1
   VAR 
      LoweringSensorPFM_Brak { S7_SetPoint := 'False'} : "Sensor_sticking_checker";   // датчик приопускания пакета пфм брака
      PFM_brak_boardcounter : "Sensor_sticking_checker";   // датчик счета доски на пфм брака
   END_VAR


BEGIN
	#LoweringSensorPFM_Brak(SensorSig:= "B22.6",
	                        StickCondition:= "ALG".Auto_defect AND NOT "ПФМ Брака_DB".LiftPushingPacket AND "ПФМ Брака_DB".HodVil,
	                        Reset:= "S76.2",
	                        Stick_time:=T#20s);
	
	#PFM_brak_boardcounter(SensorSig:="FC 22.7",
	                       StickCondition:= "ALG".Auto_defect AND "IM".M_334_Layer_set_conv.onOutFWD,
	                       Reset:="S76.2",
	                       Stick_time:=T#10s);
	
	
END_FUNCTION_BLOCK

FUNCTION_BLOCK "Sensor_sticking_checker"
{ S7_Optimized_Access := 'FALSE' }
AUTHOR : Aspir
VERSION : 0.1
   VAR_INPUT 
      SensorSig : Bool;
      StickCondition : Bool;
      Reset : Bool;
      Stick_time : Time;
   END_VAR

   VAR_OUTPUT 
      AlarmStickingSensor : Bool;
   END_VAR

   VAR 
      Stick_timer {InstructionName := 'TON'; LibVersion := '1.0'; S7_SetPoint := 'False'} : TON;
   END_VAR


BEGIN
	#Stick_timer(IN:=#SensorSig AND #StickCondition,
	             PT:=#Stick_time);
	
	#AlarmStickingSensor := (#AlarmStickingSensor OR #Stick_timer.Q) AND NOT #Reset;
	
END_FUNCTION_BLOCK

FUNCTION_BLOCK "SensorStartUp_checker"
{ S7_Optimized_Access := 'FALSE' }
AUTHOR : Aspir
VERSION : 0.1

BEGIN
END_FUNCTION_BLOCK

DATA_BLOCK "BobDropper_CNTL_DB"   // DB26
AUTHOR : Aspir
VERSION : 0.1
// stored: AutoNumber true, InstanceOfName BobDropper_CNTL, InstanceOfType FB
"BobDropper_CNTL"
BEGIN
END_DATA_BLOCK

DATA_BLOCK "CNT_CTRL_1"   // DB20
// stored: AutoNumber false, InstanceOfName CNT_CHANTYPE1, OfSystemLibElement CNT_CHANTYPE1, OfSystemLibVersion 1.0
"CNT_CHANTYPE1"
   // VAR RETAIN
   //    AR1_BUFFER : DWord;
   //    FP : Byte;
   //    RESERVED : Byte;
   //    MOD_ADR : Word := 544;
   //    CH_ADR : DWord := P#544.0;
   //    U_D_LGTH : Byte := 16#0;
   //    A_BYTE_0 : Byte;
   //    LOAD_VAL : DInt := 0;
   //    CMP_V1 : DInt;
   //    CMP_V2 : DInt;
   //    A_BIT0_0 : Bool;
   //    TFB : Bool;
   //    A_BIT0_2 : Bool;
   //    A_BIT0_3 : Bool;
   //    A_BIT0_4 : Bool;
   //    A_BIT0_5 : Bool;
   //    A_BIT0_6 : Bool;
   //    A_BIT0_7 : Bool;
   //    ENSET_UP : Bool;
   //    ENSET_DN : Bool;
   //    A_BIT1_2 : Bool;
   //    A_BIT1_3 : Bool;
   //    A_BIT1_4 : Bool;
   //    A_BIT1_5 : Bool;
   //    A_BIT1_6 : Bool;
   //    A_BIT1_7 : Bool;
   //    CTRL_DO0 : Bool;
   //    CTRL_DO1 : Bool;
   //    A_BIT2_2 : Bool;
   //    A_BIT2_3 : Bool;
   //    A_BIT2_4 : Bool;
   //    A_BIT2_5 : Bool;
   //    A_BIT2_6 : Bool;
   //    A_BIT2_7 : Bool;
   //    A_BIT3_0 : Bool;
   //    A_BIT3_1 : Bool;
   //    A_BIT3_2 : Bool;
   //    A_BIT3_3 : Bool;
   //    A_BIT3_4 : Bool;
   //    A_BIT3_5 : Bool;
   //    A_BIT3_6 : Bool;
   //    A_BIT3_7 : Bool;
   //    LATCH_LOAD : DInt;
   //    ACT_CNTV : DInt;
   //    DA_ERR_W : Word;
   //    OT_ERR_B : Byte;
   //    E_BIT0_0 : Bool;
   //    STS_TFB : Bool;
   //    DIAG : Bool;
   //    E_BIT0_3 : Bool;
   //    DATA_ERR : Bool;
   //    E_BIT0_5 : Bool;
   //    E_BIT0_6 : Bool;
   //    PARA : Bool;
   //    E_BYTE_0 : Byte;
   //    STS_RUN : Bool;
   //    STS_DIR : Bool := false;
   //    STS_ZERO : Bool;
   //    STS_OFLW : Bool;
   //    STS_UFLW : Bool;
   //    STS_SYNC : Bool;
   //    STS_GATE : Bool := false;
   //    STS_SW_G : Bool := false;
   //    STS_SET : Bool;
   //    STS_LATCH : Bool;
   //    STS_STA : Bool;
   //    STS_STP : Bool;
   //    STS_CMP1 : Bool;
   //    STS_CMP2 : Bool;
   //    STS_COMP1 : Bool;
   //    STS_COMP2 : Bool;
   //    E_BIT3_0 : Bool;
   //    E_BIT3_1 : Bool;
   //    E_BIT3_2 : Bool;
   //    E_BIT3_3 : Bool;
   //    E_BIT3_4 : Bool;
   //    E_BIT3_5 : Bool;
   //    E_BIT3_6 : Bool;
   //    E_BIT3_7 : Bool;
   //    ACT_CMP1 : DInt;
   //    ACT_CMP2 : DInt;
   //    MDL_DEFECT : Bool;
   //    INT_FAULT : Bool;
   //    EXT_FAULT : Bool;
   //    PNT_INFO : Bool;
   //    EXT_VOLTAGE : Bool;
   //    FLD_CONNCTR : Bool;
   //    NO_CONFIG : Bool;
   //    CONFIG_ERR : Bool;
   //    MDL_TYPE : Byte;
   //    SUB_MDL_ERR : Bool;
   //    COMM_FAULT : Bool;
   //    MDL_STOP : Bool;
   //    WTCH_DOG_FLT : Bool;
   //    INT_PS_FLT : Bool;
   //    PRIM_BATT_FLT : Bool;
   //    BCKUP_BATT_FLT : Bool;
   //    RESERVED_2 : Bool;
   //    RACK_FLT : Bool;
   //    PROC_FLT : Bool;
   //    EPROM_FLT : Bool;
   //    RAM_FLT : Bool;
   //    ADU_FLT : Bool;
   //    FUSE_FLT : Bool;
   //    HW_INTR_FLT : Bool;
   //    RESERVED_3 : Bool;
   //    CH_TYPE : Byte;
   //    LGTH_DIA : Byte;
   //    CH_NO : Byte;
   //    GRP_ERR1 : Bool;
   //    GRP_ERR2 : Bool;
   //    D_BIT7_2 : Bool;
   //    D_BIT7_3 : Bool;
   //    D_BIT7_4 : Bool;
   //    D_BIT7_5 : Bool;
   //    D_BIT7_6 : Bool;
   //    D_BIT7_7 : Bool;
   //    CH1_SIGA : Bool;
   //    CH1_SIGB : Bool;
   //    CH1_SIGZ : Bool;
   //    CH1_BETW : Bool;
   //    CH1_5V2 : Bool;
   //    D_BIT8_5 : Bool;
   //    D_BIT8_6 : Bool;
   //    D_BIT8_7 : Bool;
   //    D_BYTE9 : Byte;
   //    CH2_SIGA : Bool;
   //    CH2_SIGB : Bool;
   //    CH2_SIGZ : Bool;
   //    CH2_BETW : Bool;
   //    CH2_5V2 : Bool;
   //    D_BIT10_5 : Bool;
   //    D_BIT10_6 : Bool;
   //    D_BIT10_7 : Bool;
   //    D_BYTE11 : Byte;
   //    D_BYTE12 : Byte;
   //    D_BYTE13 : Byte;
   //    D_BYTE14 : Byte;
   //    D_BYTE15 : Byte;
   // END_VAR
BEGIN
END_DATA_BLOCK

DATA_BLOCK "Counter_1_DB"   // DB16
AUTHOR : PSIfunc
VERSION : 0.1
// stored: AutoNumber true, InstanceOfName Counter_1, InstanceOfType FB
"Counter_1"
BEGIN
END_DATA_BLOCK

DATA_BLOCK "DGI"   // DB2
VERSION : 0.1
// stored: AutoNumber true, InstanceOfName GetDiskretInputs, InstanceOfType FB
"GetDiskretInputs"
BEGIN
END_DATA_BLOCK

DATA_BLOCK "DynamicLayer_CNTL_DB"   // DB24
AUTHOR : Aspir
VERSION : 0.1
// stored: AutoNumber true, InstanceOfName DynamicLayer_CNTL, InstanceOfType FB
"DynamicLayer_CNTL"
BEGIN
END_DATA_BLOCK

DATA_BLOCK "EvaluationZoneThrowOFF_DB"   // DB22
VERSION : 0.1
// stored: AutoNumber true, InstanceOfName EvaluationZoneThrowOFF, InstanceOfType FB
"EvaluationZoneThrowOFF"
BEGIN
END_DATA_BLOCK

DATA_BLOCK "FB_Gasket_Carousel_DB"   // DB32
VERSION : 0.1
// stored: AutoNumber true, InstanceOfName FB_Gasket_Carousel, InstanceOfType FB
"FB_Gasket_Carousel"
BEGIN
END_DATA_BLOCK

DATA_BLOCK "FB_Load_Zone_DB"   // DB30
VERSION : 0.1
// stored: AutoNumber true, InstanceOfName FB_Load_Zone, InstanceOfType FB
"FB_Load_Zone"
BEGIN
END_DATA_BLOCK

DATA_BLOCK "FB_Ramp_DB"   // DB15
VERSION : 0.1
// stored: AutoNumber true, InstanceOfName FB_Ramp, InstanceOfType FB
"FB_Ramp"
BEGIN
END_DATA_BLOCK

DATA_BLOCK "FB_Rollout_Zone_DB"   // DB31
VERSION : 0.1
// stored: AutoNumber true, InstanceOfName FB_Rollout_Zone, InstanceOfType FB
"FB_Rollout_Zone"
BEGIN
END_DATA_BLOCK

DATA_BLOCK "FB_SensLine_DB"   // DB17
AUTHOR : Aspir
VERSION : 0.1
// stored: AutoNumber true, InstanceOfName FB_SensLine, InstanceOfType FB
"FB_SensLine"
BEGIN
END_DATA_BLOCK

DATA_BLOCK "HS"   // DB21
VERSION : 0.1
// stored: AutoNumber true, InstanceOfName FB_HydroStations, InstanceOfType FB
"FB_HydroStations"
BEGIN
END_DATA_BLOCK

DATA_BLOCK "IM"   // DB10
VERSION : 0.1
// stored: AutoNumber true, InstanceOfName FB_IM, InstanceOfType FB
"FB_IM"
BEGIN
END_DATA_BLOCK

DATA_BLOCK "IM_PFM"   // DB14
VERSION : 0.1
// stored: AutoNumber true, InstanceOfName FB_IM_PFM, InstanceOfType FB
"FB_IM_PFM"
BEGIN
   M_233_Fork_PFM.SpeedOn := 15.0;
   M_233_Fork_PFM.SpeedOnLow := 10.0;
   M_233_Fork_PFM.SpeedOff := 15.0;
   M_233_Fork_PFM.SpeedOffLow := 10.0;
END_DATA_BLOCK

DATA_BLOCK "IM_Rout"   // DB23
VERSION : 0.1
// stored: AutoNumber true, InstanceOfName FB_IM_Rout, InstanceOfType FB
"FB_IM_Rout"
BEGIN
END_DATA_BLOCK

DATA_BLOCK "KeyFazer_CNTL_DB"   // DB28
AUTHOR : Aspir
VERSION : 0.1
// stored: AutoNumber true, InstanceOfName KeyFazer_CNTL, InstanceOfType FB
"KeyFazer_CNTL"
BEGIN
END_DATA_BLOCK

DATA_BLOCK "KeyFazer_Counter_DB"   // DB29
AUTHOR : Aspir
VERSION : 0.1
// stored: AutoNumber true, InstanceOfName KeyFazer_Counter, InstanceOfType FB
"KeyFazer_Counter"
BEGIN
END_DATA_BLOCK

DATA_BLOCK "MovableBoard_CTRL_DB"   // DB13
VERSION : 0.1
// stored: AutoNumber true, InstanceOfName MovableBoard_CTRL, InstanceOfType FB
"MovableBoard_CTRL"
BEGIN
END_DATA_BLOCK

DATA_BLOCK "QueueController_DB"   // DB11
AUTHOR : Aspir
VERSION : 0.1
// stored: AutoNumber true, InstanceOfName QueueController, InstanceOfType FB
"QueueController"
BEGIN
END_DATA_BLOCK

DATA_BLOCK "SensLine_SigAdapter_DB"   // DB27
VERSION : 0.1
// stored: AutoNumber true, InstanceOfName SensLine_SigAdapter, InstanceOfType FB
"SensLine_SigAdapter"
BEGIN
END_DATA_BLOCK

DATA_BLOCK "SensorLine_Clogging_DB"   // DB25
VERSION : 0.1
// stored: AutoNumber true, InstanceOfName SensorLine_Clogging, InstanceOfType FB
"SensorLine_Clogging"
BEGIN
END_DATA_BLOCK

DATA_BLOCK "ServDB"   // DB5
VERSION : 0.1
// stored: AutoNumber true, InstanceOfName FB_Link_Server, InstanceOfType FB
"FB_Link_Server"
BEGIN
END_DATA_BLOCK

DATA_BLOCK "UporPFM_DB"   // DB12
VERSION : 0.1
// stored: AutoNumber true, InstanceOfName UporPFM, InstanceOfType FB
"UporPFM"
BEGIN
END_DATA_BLOCK

DATA_BLOCK "Безопасность_DB"   // DB1
VERSION : 0.1
// stored: AutoNumber true, InstanceOfName Безопасность, InstanceOfType FB
"Безопасность"
BEGIN
END_DATA_BLOCK

DATA_BLOCK "Загрузка_DB"   // DB3
VERSION : 0.1
// stored: AutoNumber true, InstanceOfName Загрузка, InstanceOfType FB
"Загрузка"
BEGIN
END_DATA_BLOCK

DATA_BLOCK "ПФМ Брака_DB"   // DB8
VERSION : 0.1
// stored: AutoNumber true, InstanceOfName ПФМ Брака, InstanceOfType FB
"ПФМ Брака"
BEGIN
END_DATA_BLOCK

DATA_BLOCK "Подача прокладки_DB"   // DB6
VERSION : 0.1
// stored: AutoNumber true, InstanceOfName Подача прокладки, InstanceOfType FB
"Подача прокладки"
BEGIN
END_DATA_BLOCK

DATA_BLOCK "Сортировка_DB"   // DB7
VERSION : 0.1
// stored: AutoNumber true, InstanceOfName Сортировка, InstanceOfType FB
"Сортировка"
BEGIN
END_DATA_BLOCK
